{attribute 'GeneratedUsingTerminal: EL3423-0000-0020'}
{attribute addProperty BoxType "EL3423-0000-0020"}
{attribute addProperty Id "Total_StatusAT %I*Total_Status_1ACE98F018Total_AdvancedAT %I*Total_Advanced_3B87F4672Total_Statistic_PowerAT %I*Total_Statistic_Power_092925BE36Total_Statistic_PQFAT %I*Total_Statistic_PQF_E024324412Total_Active_ReducedAT %I*Total_Active_Reduced_0E616AE58Total_Apparent_ReducedAT %I*Total_Apparent_Reduced_4B7F30148Total_Reactive_ReducedAT %I*Total_Reactive_Reduced_207ED80C8Total_Interval_Energy_ReducedAT %I*Total_Interval_Energy_Reduced_B0A0CDD813Total_IntervalAT %Q*Total_Interval_1578BBD41WcStateAT %I*WcState_9091E0EB2InfoDataAT %I*InfoData_94A18F5E2"}
{attribute addProperty CRC "2844660352"}
{attribute addProperty Size "110"}
TYPE EL3423_A98E1280 EXTENDS EtcSlaveTerminalBase_947E5A46 :
STRUCT
	{attribute addProperty Name "Total_Status"}
	Total_Status : Total_Status_1ACE98F0;
	{attribute addProperty Name "Total_Advanced"}
	Total_Advanced : Total_Advanced_3B87F467;
	{attribute addProperty Name "Total_Statistic_Power"}
	Total_Statistic_Power : Total_Statistic_Power_092925BE;
	{attribute addProperty Name "Total_Statistic_PQF"}
	Total_Statistic_PQF : Total_Statistic_PQF_E0243244;
	{attribute addProperty Name "Total_Active_Reduced"}
	Total_Active_Reduced : Total_Active_Reduced_0E616AE5;
	{attribute addProperty Name "Total_Apparent_Reduced"}
	Total_Apparent_Reduced : Total_Apparent_Reduced_4B7F3014;
	{attribute addProperty Name "Total_Reactive_Reduced"}
	Total_Reactive_Reduced : Total_Reactive_Reduced_207ED80C;
	{attribute addProperty Name "Total_Interval_Energy_Reduced"}
	Total_Interval_Energy_Reduced : Total_Interval_Energy_Reduced_B0A0CDD8;
	{attribute addProperty Name "Total_Interval"}
	Total_Interval : Total_Interval_1578BBD4;
	{attribute addProperty Name "WcState"}
	WcState : WcState_9091E0EB;
	{attribute addProperty Name "InfoData"}
	InfoData : InfoData_94A18F5E;
END_STRUCT
END_TYPE

(* stored: Version 1.2.0.0, ProductVersion 3.1.4024.9
   DUT EL3423_A98E1280: Id {53042a6f-0a48-46b0-8d9e-8164422dc6e2} *)
